{attribute 'hide'}
{attribute 'reflection'}
FUNCTION_BLOCK T_Integer
VAR
    Value : INT;
END_VAR

{attribute 'TcRpcEnable'}
METHOD Inc : INT
VAR_INPUT
END_VAR
Value := Value + 1;
Inc   := Value;
END_METHOD

METHOD Init
VAR_INPUT
    Value : INT;
END_VAR
THIS^.Value := Value;
END_METHOD

END_FUNCTION_BLOCK

(* stored: Version 1.1.0.1, ProductVersion 3.1.4024.12
   POU T_Integer: Id {3d96099e-d03a-0a7c-17f3-8d23f37e5358}, SpecialFunc None
   Method Inc: Id {a7bd1891-50ab-0801-2d64-d490c718e3c7}
   Method Init: Id {7deb6d59-8977-0489-2653-46330f894495} *)
